SYSTEM test_Training_02_OPC_UA
  (* Version 1.0, 2026-09-02, Franz Höpfinger, Meisterschulen am Ostbahnhof *)
  PACKAGE Training_OPC_UA_RES;
  IMPORT logiBUS::stations::Computers::C_11;
  IMPORT logiBUS::stations::Computers::C_12;
  IMPORT logiBUS::io::DI::logiBUS_DI::Input_I1;
  IMPORT logiBUS::io::DQ::logiBUS_DO::Output_Q1;
  IMPORT VV::const::OPC_UA::myOpcUaAddresses::Q1_LOCAL_READ;
  IMPORT VV::const::OPC_UA::myOpcUaAddresses::Q1_REMOTE_WRITE;
  APPLICATION App_OPC_UA_RES
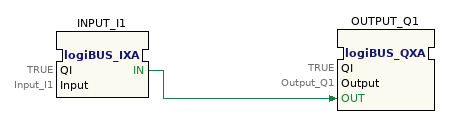
    FBS
      INPUT_I1 : logiBUS::io::DI::logiBUS_IXA(QI := TRUE, Input := Input_I1);
      OUTPUT_Q1 : logiBUS::io::DQ::logiBUS_QXA(QI := TRUE, Output := Output_Q1);
    END_FBS
    ADAPTER_CONNECTIONS
      INPUT_I1.IN TO OUTPUT_Q1.OUT;
    END_CONNECTIONS
  END_APPLICATION
  DEVICE FORTE_PC_A : iec61499::system::FORTE_PC(MGR_ID := C_11 (* Device manager socket ID *))
    {SET_ATTRIBUTE(Profile, HOLOBLOC)}
    RESOURCE EMB_RES_A : iec61499::system::EMB_RES
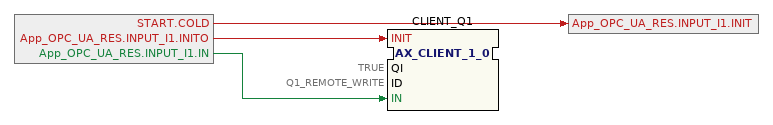
      FBS
        CLIENT_Q1 : adapter::net::AX_CLIENT_1_0(QI := TRUE, ID := Q1_REMOTE_WRITE);
      END_FBS
      EVENT_CONNECTIONS
        START.COLD TO App_OPC_UA_RES.INPUT_I1.INIT;
        App_OPC_UA_RES.INPUT_I1.INITO TO CLIENT_Q1.INIT;
      END_CONNECTIONS
      ADAPTER_CONNECTIONS
        App_OPC_UA_RES.INPUT_I1.IN TO CLIENT_Q1.IN;
      END_CONNECTIONS
    END_RESOURCE
  END_DEVICE
  DEVICE FORTE_PC_B : iec61499::system::FORTE_PC(MGR_ID := C_12 (* Device manager socket ID *))
    {SET_ATTRIBUTE(Profile, HOLOBLOC)}
    RESOURCE EMB_RES_B : iec61499::system::EMB_RES
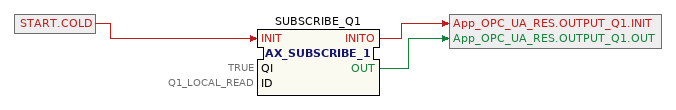
      FBS
        SUBSCRIBE_Q1 : adapter::net::AX_SUBSCRIBE_1(QI := TRUE, ID := Q1_LOCAL_READ);
      END_FBS
      EVENT_CONNECTIONS
        START.COLD TO SUBSCRIBE_Q1.INIT;
        SUBSCRIBE_Q1.INITO TO App_OPC_UA_RES.OUTPUT_Q1.INIT;
      END_CONNECTIONS
      ADAPTER_CONNECTIONS
        SUBSCRIBE_Q1.OUT TO App_OPC_UA_RES.OUTPUT_Q1.OUT;
      END_CONNECTIONS
    END_RESOURCE
  END_DEVICE
  MAPPINGS
    App_OPC_UA_RES.INPUT_I1 ON FORTE_PC_A.EMB_RES_A;
    App_OPC_UA_RES.OUTPUT_Q1 ON FORTE_PC_B.EMB_RES_B;
  END_MAPPINGS
  SEGMENTS
    Ethernet : iec61499::system::Ethernet;
  END_SEGMENTS
  LINKS
    FORTE_PC_A => Ethernet;
    FORTE_PC_B => Ethernet;
  END_LINKS
END_SYSTEM
